KUKA KRL data list: wkz3_an.dat

&ACCESS RVO2
&REL 176
&COMMENT PEGA_GRIPPER_ACCELO
&PARAM DISKPATH = KRC:\R1\Program\WKZ
DEFDAT  wkz3_an
;FOLD EXTERNAL DECLARATIONS;%{PE}%MKUKATPBASIS,%CEXT,%VCOMMON,%P
;FOLD BASISTECH EXT;%{PE}%MKUKATPBASIS,%CEXT,%VEXT,%P
EXT  BAS (BAS_COMMAND  :IN,REAL  :IN )
DECL INT SUCCESS
;ENDFOLD (BASISTECH EXT)
;FOLD USER EXT;%{E}%MKUKATPUSER,%CEXT,%VEXT,%P
;Make your modifications here
;ENDFOLD (USER EXT)
;ENDFOLD (EXTERNAL DECLARATIONS)

;# ============ START PATH : wkz3_an =============
DECL FDAT Fnew_wkz3_an_p11={TOOL_NO 8,BASE_NO 2,IPO_FRAME #BASE,POINT2[] " ",TQ_STATE FALSE}
DECL PDAT PP_OLP1={VEL 100.0,ACC 100.0,APO_DIST 0.0,APO_MODE #CPTP}
DECL E6POS Xnew_wkz3_an_p11={X -2369.50391,Y 3754.82593,Z 418.015991,A 152.721802,B -13.0292997,C 137.894104,S 2,T 2}
DECL FDAT Fnew_wkz3_an_p3={TOOL_NO 8,BASE_NO 0,IPO_FRAME #BASE,POINT2[] " "}
DECL PDAT PP_OLP2={VEL 50.0,ACC 100.0,APO_DIST 0.0,APO_MODE #CPTP}
DECL E6POS Xnew_wkz3_an_p3={X 285.191986,Y -1942.47998,Z 150.375,A 11.8746996,B 8.36009979,C 151.334,S 2,T 2}
DECL FDAT Fnew_wkz3_an_p4={TOOL_NO 8,BASE_NO 0,IPO_FRAME #BASE,POINT2[] " ",TQ_STATE FALSE}
DECL E6POS Xnew_wkz3_an_p4={X 280.436005,Y -2032.76697,Z -7.78399992,A 11.8758001,B 8.36009979,C 151.335403,S 2,T 2}
DECL LDAT LL_OLP1={VEL 0.100000001,ACC 100.0,APO_DIST 0.0,APO_FAC 0.0,ORI_TYP #VAR,CIRC_TYP #BASE,JERK_FAC 50.0}
DECL FDAT Fnew_wkz3_an_p5={TOOL_NO 8,BASE_NO 0,IPO_FRAME #BASE,POINT2[] " "}
DECL E6POS Xnew_wkz3_an_p5={X 279.769714,Y -2045.62402,Z -30.3428097,A 11.8758698,B 8.35940933,C 151.336304,S 18,T 2,E1 0.0,E2 0.0,E3 0.0,E4 0.0,E5 0.0,E6 0.0}
DECL LDAT LL_OLP2={VEL 0.100000001,ACC 100.0,APO_DIST 0.0,APO_FAC 0.0,ORI_TYP #VAR,CIRC_TYP #BASE,JERK_FAC 50.0}
DECL FDAT Fnew_wkz3_an_p13={TOOL_NO 3,BASE_NO 0,IPO_FRAME #BASE,POINT2[] " "}
DECL E6POS Xnew_wkz3_an_p13={X 320.731903,Y -1358.099,Z -453.487305,A -1.25453806,B 1.00949597,C -179.808502,S 18,T 2,E1 0.0,E2 0.0,E3 0.0,E4 0.0,E5 0.0,E6 0.0}
DECL LDAT LL_OLP3={VEL 0.100000001,ACC 100.0,APO_DIST 100.0,APO_FAC 50.0,ORI_TYP #VAR,CIRC_TYP #BASE,JERK_FAC 50.0}
DECL FDAT Fnew_wkz3_an_p6={TOOL_NO 3,BASE_NO 0,IPO_FRAME #BASE,POINT2[] " ",TQ_STATE FALSE}
DECL E6POS Xnew_wkz3_an_p6={X 320.2789,Y -1358.29297,Z 76.6145401,A -1.25866401,B 1.00914299,C -179.787201,S 18,T 2,E1 0.0,E2 0.0,E3 0.0,E4 0.0,E5 0.0,E6 0.0}
DECL LDAT LL_OLP4={VEL 0.100000001,ACC 100.0,APO_DIST 100.0,APO_FAC 50.0,ORI_TYP #VAR,CIRC_TYP #BASE,JERK_FAC 50.0}
DECL FDAT Fnew_wkz3_an_p16={TOOL_NO 3,BASE_NO 0,IPO_FRAME #BASE,POINT2[] " "}
DECL E6POS Xnew_wkz3_an_p16={X 308.81601,Y -1299.86694,Z -334.415985,A -1.23179996,B 0.969600022,C -179.970398,S 2,T 2}
DECL LDAT LL_OLP5={VEL 0.400000006,ACC 40.0,APO_DIST 100.0,APO_FAC 50.0,ORI_TYP #VAR,CIRC_TYP #BASE,JERK_FAC 50.0}
DECL FDAT Fnew_wkz3_an_p17={TOOL_NO 3,BASE_NO 0,IPO_FRAME #BASE,POINT2[] " "}
DECL E6POS Xnew_wkz3_an_p17={X 246.035004,Y -1298.23804,Z -267.673004,A -1.22860003,B 5.79850006,C -179.955399,S 2,T 2}
DECL LDAT LL_OLP6={VEL 0.100000001,ACC 100.0,APO_DIST 100.0,APO_FAC 50.0,ORI_TYP #VAR,CIRC_TYP #BASE,JERK_FAC 50.0}
DECL FDAT Fnew_wkz3_an_p18={TOOL_NO 3,BASE_NO 0,IPO_FRAME #BASE,POINT2[] " "}
DECL E6POS Xnew_wkz3_an_p18={X 246.768005,Y -1241.82703,Z 44.9319992,A -1.22679996,B 6.41340017,C -179.964203,S 2,T 2}
DECL LDAT LL_OLP7={VEL 0.100000001,ACC 100.0,APO_DIST 100.0,APO_FAC 50.0,ORI_TYP #VAR,CIRC_TYP #BASE,JERK_FAC 50.0}
DECL FDAT Fnew_wkz3_an_p15={TOOL_NO 3,BASE_NO 0,IPO_FRAME #BASE,POINT2[] " "}
DECL PDAT PP_OLP3={VEL 50.0,ACC 100.0,APO_DIST 0.0}
DECL E6POS Xnew_wkz3_an_p15={X 355.109985,Y -1126.28003,Z 317.824005,A -1.22809994,B 6.4151001,C -179.964706,S 2,T 2}
DECL FDAT Fnew_wkz3_an_p12={TOOL_NO 3,BASE_NO 0,IPO_FRAME #BASE,POINT2[] " "}
DECL PDAT PP_OLP4={VEL 100.0,ACC 50.0,APO_DIST 0.0}
DECL E6POS Xnew_wkz3_an_p12={X 1101.30701,Y -1142.58203,Z 1005.07397,A -29.1075001,B -30.0671005,C 172.807495,S 2,T 2}
DECL FDAT Fnew_wkz3_an_p19={TOOL_NO 3,BASE_NO 0,IPO_FRAME #BASE,POINT2[] " "}
DECL PDAT PP_OLP5={VEL 100.0,ACC 100.0,APO_DIST 0.0}
DECL E6POS Xnew_wkz3_an_p19={X 1376.82104,Y -1401.61206,Z 1623.00403,A -28.9841995,B -54.9752998,C 168.858795,S 2,T 2}
DECL E6POS XP1={X 1055.88599,Y -1502.41895,Z 1588.45996,A -71.8711777,B -60.8085899,C 178.738098,S 18,T 2,E1 0.0,E2 0.0,E3 0.0,E4 0.0,E5 0.0,E6 0.0}
DECL BASIS_SUGG_T LAST_BASIS={POINT1[] "p13                     ",POINT2[] "p13                     ",CP_PARAMS[] "CPDAT5                  ",PTP_PARAMS[] "PDAT9                   ",CONT[] "C_PTP                   ",CP_VEL[] "0.1                     ",PTP_VEL[] "100                     ",SYNC_PARAMS[] "SYNCDAT                 ",SPL_NAME[] "S0                      "}
DECL FDAT FP1={TOOL_NO 8,BASE_NO 0,IPO_FRAME #BASE,POINT2[] " ",TQ_STATE FALSE}
DECL PDAT PPDAT1={VEL 100.0,ACC 100.0,APO_DIST 100.0,APO_MODE #CPTP,GEAR_JERK 50.0}
DECL PDAT PPDAT2={VEL 100.0,ACC 100.0,APO_DIST 100.0,GEAR_JERK 50.0}
DECL E6POS XP2={X 1055.88794,Y -1502.41699,Z 1588.45105,A -71.872261,B -60.8076706,C 178.739105,S 18,T 2,E1 0.0,E2 0.0,E3 0.0,E4 0.0,E5 0.0,E6 0.0}
DECL FDAT Fp2={TOOL_NO 8,BASE_NO 0,IPO_FRAME #BASE,POINT2[] " ",TQ_STATE FALSE}
DECL PDAT PPDAT3={VEL 100.0,ACC 100.0,APO_DIST 0.0,APO_MODE #CPTP,GEAR_JERK 50.0}
DECL E6POS XP3={X 609.982727,Y -1742.26501,Z 928.062012,A -27.3751602,B -12.9938002,C 137.779007,S 18,T 2,E1 0.0,E2 0.0,E3 0.0,E4 0.0,E5 0.0,E6 0.0}
DECL FDAT Fp3={TOOL_NO 8,BASE_NO 0,IPO_FRAME #BASE,POINT2[] " ",TQ_STATE FALSE}
DECL PDAT PPDAT4={VEL 100.0,ACC 100.0,APO_DIST 100.0,APO_MODE #CPTP,GEAR_JERK 50.0}
DECL E6POS XP4={X -2046.27698,Y 3954.58105,Z -360.438812,A -167.992798,B 8.26109791,C 151.400101,S 18,T 2,E1 0.0,E2 0.0,E3 0.0,E4 0.0,E5 0.0,E6 0.0}
DECL FDAT Fp4={TOOL_NO 8,BASE_NO 2,IPO_FRAME #BASE,POINT2[] " ",TQ_STATE FALSE}
DECL PDAT PPDAT5={VEL 100.0,ACC 100.0,APO_DIST 0.0,APO_MODE #CPTP,GEAR_JERK 50.0}
DECL E6POS XP5={X 280.258514,Y -2033.65906,Z -9.63728237,A 11.8786201,B 8.35937405,C 151.335907,S 18,T 2,E1 0.0,E2 0.0,E3 0.0,E4 0.0,E5 0.0,E6 0.0}
DECL FDAT Fp5={TOOL_NO 8,BASE_NO 0,IPO_FRAME #BASE,POINT2[] " ",TQ_STATE FALSE}
DECL LDAT LCPDAT1={VEL 2.0,ACC 100.0,APO_DIST 100.0,APO_FAC 50.0,AXIS_VEL 100.0,AXIS_ACC 100.0,ORI_TYP #VAR,CIRC_TYP #BASE,JERK_FAC 50.0,GEAR_JERK 50.0,EXAX_IGN 0}
DECL E6POS XP6={X 279.745209,Y -2046.13696,Z -31.2646408,A 11.8763199,B 8.35891533,C 151.337204,S 18,T 2,E1 0.0,E2 0.0,E3 0.0,E4 0.0,E5 0.0,E6 0.0}
DECL FDAT Fp6={TOOL_NO 8,BASE_NO 0,IPO_FRAME #BASE,POINT2[] " ",TQ_STATE FALSE}
DECL LDAT LCPDAT2={VEL 2.0,ACC 100.0,APO_DIST 100.0,APO_FAC 50.0,AXIS_VEL 100.0,AXIS_ACC 100.0,ORI_TYP #VAR,CIRC_TYP #BASE,JERK_FAC 50.0,GEAR_JERK 50.0,EXAX_IGN 0}
DECL E6POS XP7={X 320.729401,Y -1358.09802,Z -453.486786,A -1.25442803,B 1.00959301,C -179.808395,S 18,T 2,E1 0.0,E2 0.0,E3 0.0,E4 0.0,E5 0.0,E6 0.0}
DECL FDAT Fp7={TOOL_NO 3,BASE_NO 0,IPO_FRAME #BASE,POINT2[] " ",TQ_STATE FALSE}
DECL LDAT LCPDAT3={VEL 2.0,ACC 100.0,APO_DIST 100.0,APO_FAC 50.0,AXIS_VEL 100.0,AXIS_ACC 100.0,ORI_TYP #VAR,CIRC_TYP #BASE,JERK_FAC 50.0,GEAR_JERK 50.0,EXAX_IGN 0}
DECL E6POS XP8={X 320.276886,Y -1358.29004,Z 76.6149673,A -1.258533,B 1.00919104,C -179.787094,S 18,T 2,E1 0.0,E2 0.0,E3 0.0,E4 0.0,E5 0.0,E6 0.0}
DECL FDAT Fp8={TOOL_NO 3,BASE_NO 0,IPO_FRAME #BASE,POINT2[] " ",TQ_STATE FALSE}
DECL LDAT LCPDAT4={VEL 2.0,ACC 100.0,APO_DIST 100.0,APO_FAC 50.0,AXIS_VEL 100.0,AXIS_ACC 100.0,ORI_TYP #VAR,CIRC_TYP #BASE,JERK_FAC 50.0,GEAR_JERK 50.0,EXAX_IGN 0}
DECL E6POS XP9={X 246.780502,Y -1241.81396,Z 44.9335594,A -1.22680402,B 6.41300392,C -179.963593,S 18,T 2,E1 0.0,E2 0.0,E3 0.0,E4 0.0,E5 0.0,E6 0.0}
DECL FDAT Fp9={TOOL_NO 3,BASE_NO 0,IPO_FRAME #BASE,POINT2[] " ",TQ_STATE FALSE}
DECL LDAT LCPDAT5={VEL 2.0,ACC 100.0,APO_DIST 100.0,APO_FAC 50.0,AXIS_VEL 100.0,AXIS_ACC 100.0,ORI_TYP #VAR,CIRC_TYP #BASE,JERK_FAC 50.0,GEAR_JERK 50.0,EXAX_IGN 0}
DECL E6POS XP10={X 355.111511,Y -1126.27197,Z 317.824188,A -1.22783005,B 6.41505194,C -179.964096,S 18,T 2,E1 0.0,E2 0.0,E3 0.0,E4 0.0,E5 0.0,E6 0.0}
DECL FDAT Fp10={TOOL_NO 3,BASE_NO 0,IPO_FRAME #BASE,POINT2[] " ",TQ_STATE FALSE}
DECL PDAT PPDAT6={VEL 100.0,ACC 50.0,APO_DIST 100.0,APO_MODE #CPTP,GEAR_JERK 50.0}
DECL E6POS XP11={X 1101.30798,Y -1142.57996,Z 1005.07001,A -29.1077003,B -30.0667191,C 172.807999,S 18,T 2,E1 0.0,E2 0.0,E3 0.0,E4 0.0,E5 0.0,E6 0.0}
DECL FDAT Fp11={TOOL_NO 3,BASE_NO 0,IPO_FRAME #BASE,POINT2[] " ",TQ_STATE FALSE}
DECL PDAT PPDAT7={VEL 100.0,ACC 50.0,APO_DIST 100.0,APO_MODE #CPTP,GEAR_JERK 50.0}
DECL E6POS XP12={X 1376.823,Y -1401.60999,Z 1623.0,A -28.9847107,B -54.9749184,C 168.859406,S 18,T 2,E1 0.0,E2 0.0,E3 0.0,E4 0.0,E5 0.0,E6 0.0}
DECL FDAT Fp12={TOOL_NO 3,BASE_NO 0,IPO_FRAME #BASE,POINT2[] " ",TQ_STATE FALSE}
DECL PDAT PPDAT8={VEL 100.0,ACC 50.0,APO_DIST 0.0,APO_MODE #CPTP,GEAR_JERK 50.0}
DECL E6POS XP13={X 270.12619,Y -1985.93506,Z 129.894501,A 11.9555597,B 10.6837397,C 151.723404,S 18,T 2,E1 0.0,E2 0.0,E3 0.0,E4 0.0,E5 0.0,E6 0.0}
DECL FDAT Fp13={TOOL_NO 8,BASE_NO 0,IPO_FRAME #BASE,POINT2[] " ",TQ_STATE FALSE}
DECL PDAT PPDAT9={VEL 100.0,ACC 100.0,APO_DIST 100.0,APO_MODE #CPTP,GEAR_JERK 50.0}
ENDDAT
